FUNCTION_BLOCK FB_Variables
VAR
    normalVar : INT := 0;
END_VAR

VAR_TEMP
    tempVar : INT:=0;
END_VAR

normalVar := normalVar + 1;
tempVar := tempVar + 1;
// staticVar := staticVar + 1;

END_FUNCTION_BLOCK

(* stored: Version 1.1.0.1, ProductVersion 3.1.4024.16
   POU FB_Variables: Id {78fb358d-1306-48d7-b404-886837caf5ee}, SpecialFunc None *)
